INTERFACE I_LogPublisher EXTENDS I_Base

METHOD Subscribe : BOOL
VAR_INPUT
	Logger : I_Logger;
END_VAR
END_METHOD

METHOD Unsubscribe : BOOL
VAR_INPUT
	Logger : I_Logger;
END_VAR
END_METHOD

END_INTERFACE

(* stored: Version 1.1.0.1, ProductVersion 3.1.4026.18
   Itf I_LogPublisher: Id {ea9d2ea5-43f4-4650-af40-51c63840987d}
   Method Subscribe: Id {74e714b6-6b9c-4109-8cf4-bb7075dbf021}
   Method Unsubscribe: Id {c8393ae7-2496-47c0-adeb-8f4bdc3ac4ba} *)
